FUNCTION EMPTYSTR2 : BOOL
VAR_INPUT
	pSTR : POINTER TO STRING;
END_VAR

EMPTYSTR2 := DELETE2(pSTR,pSTR,SIZEOF(pSTR^),LEN2(pSTR),1);

END_FUNCTION

(* stored: Version 1.1.0.1, ProductVersion 3.1.4024.12
   POU EMPTYSTR2: Id {5389afbc-b10d-4582-9ce2-03d3110283b8}, SpecialFunc None *)
